PROGRAM GranulationProcess
VAR
	fbGranulationProcess : FB_GranulationProcess;
END_VAR

ACT_Granulation();

ACTION ACT_Granulation:
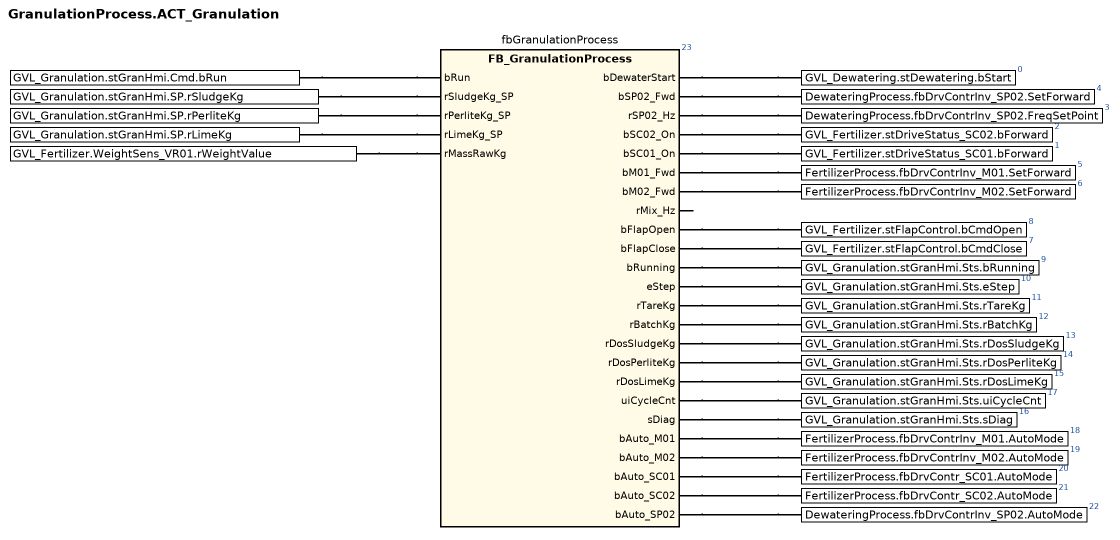
GVL_Dewatering.stDewatering.bStart := fbGranulationProcess.bDewaterStart;
GVL_Fertilizer.stDriveStatus_SC01.bForward := fbGranulationProcess.bSC01_On;
GVL_Fertilizer.stDriveStatus_SC02.bForward := fbGranulationProcess.bSC02_On;
DewateringProcess.fbDrvContrInv_SP02.FreqSetPoint := fbGranulationProcess.rSP02_Hz;
DewateringProcess.fbDrvContrInv_SP02.SetForward := fbGranulationProcess.bSP02_Fwd;
FertilizerProcess.fbDrvContrInv_M01.SetForward := fbGranulationProcess.bM01_Fwd;
FertilizerProcess.fbDrvContrInv_M02.SetForward := fbGranulationProcess.bM02_Fwd;
GVL_Fertilizer.stFlapControl.bCmdClose := fbGranulationProcess.bFlapClose;
GVL_Fertilizer.stFlapControl.bCmdOpen := fbGranulationProcess.bFlapOpen;
GVL_Granulation.stGranHmi.Sts.bRunning := fbGranulationProcess.bRunning;
GVL_Granulation.stGranHmi.Sts.eStep := fbGranulationProcess.eStep;
GVL_Granulation.stGranHmi.Sts.rTareKg := fbGranulationProcess.rTareKg;
GVL_Granulation.stGranHmi.Sts.rBatchKg := fbGranulationProcess.rBatchKg;
GVL_Granulation.stGranHmi.Sts.rDosSludgeKg := fbGranulationProcess.rDosSludgeKg;
GVL_Granulation.stGranHmi.Sts.rDosPerliteKg := fbGranulationProcess.rDosPerliteKg;
GVL_Granulation.stGranHmi.Sts.rDosLimeKg := fbGranulationProcess.rDosLimeKg;
GVL_Granulation.stGranHmi.Sts.sDiag := fbGranulationProcess.sDiag;
GVL_Granulation.stGranHmi.Sts.uiCycleCnt := fbGranulationProcess.uiCycleCnt;
FertilizerProcess.fbDrvContrInv_M01.AutoMode := fbGranulationProcess.bAuto_M01;
FertilizerProcess.fbDrvContrInv_M02.AutoMode := fbGranulationProcess.bAuto_M02;
FertilizerProcess.fbDrvContr_SC01.AutoMode := fbGranulationProcess.bAuto_SC01;
FertilizerProcess.fbDrvContr_SC02.AutoMode := fbGranulationProcess.bAuto_SC02;
DewateringProcess.fbDrvContrInv_SP02.AutoMode := fbGranulationProcess.bAuto_SP02;
fbGranulationProcess(
    bRun := GVL_Granulation.stGranHmi.Cmd.bRun,
    rSludgeKg_SP := GVL_Granulation.stGranHmi.SP.rSludgeKg,
    rPerliteKg_SP := GVL_Granulation.stGranHmi.SP.rPerliteKg,
    rLimeKg_SP := GVL_Granulation.stGranHmi.SP.rLimeKg,
    rMassRawKg := GVL_Fertilizer.WeightSens_VR01.rWeightValue); // FB_GranulationProcess
END_ACTION

END_PROGRAM

(* stored: Version 1.1.0.1, ProductVersion 3.1.4024.15
   POU GranulationProcess: Id {def867bb-983f-4959-9a14-9e1c1faa37ca}, SpecialFunc None
   Action ACT_Granulation: Id {d2edd858-827c-48fc-b4ba-6e3afe06934a} *)
